// TIA Portal V18 export
TYPE "UDT_Recipe_ATEQ"
   STRUCT
      Pressure_UL : Real;
      Pressure_LL : Real;
      Leak_UL : Real;
      Leak_LL : Real;
      PosPressureProgNo : Int;
      NegPressureProgNo : Int;
   END_STRUCT;
END_TYPE
